FUNCTION_BLOCK Station IMPLEMENTS IStation
VAR_INPUT
END_VAR
VAR_OUTPUT
END_VAR
VAR
	_Clear : BOOL;
	_Complete : BOOL;
	_Operating : BOOL;
	_Ready : BOOL;
	_Positions : ARRAY[1..4] OF MC_LREAL;
	NumberOfPositions : INT;
	AssignedPositions : INT := 1;
	StationMovers : INT;
	_OperationTime : TIME := T#1S;
	Operation : ton;
	_HasMover : BOOL;
END_VAR

IF _HasMover THEN
	_Operating := TRUE;
	_Clear := FALSE;
	_Ready := FALSE;
	Operation.IN := TRUE;
	IF Operation.Q THEN
		_Complete := TRUE;
		IF StationMovers = 0 THEN
			_HasMover := FALSE;
			Operation.IN := FALSE;
		END_IF
	END_IF
ELSE
	_Complete := FALSE;
	_Clear := TRUE;
	_Operating := FALSE;
	_Ready := TRUE;
END_IF

Operation(PT := _OperationTime);

{warning 'add method implementation '}
METHOD HasMover : BOOL
StationMovers := StationMovers + 1;
IF StationMovers = NumberOfPositions THEN
	_HasMover := TRUE;
END_IF
END_METHOD

{warning 'add method implementation '}
METHOD IsClear : BOOL
IsClear := _Clear;
END_METHOD

{warning 'add method implementation '}
METHOD isComplete : BOOL
isComplete := _Complete;
END_METHOD

{warning 'add method implementation '}
METHOD IsOperating : BOOL
IsOperating := _Operating;
END_METHOD

{warning 'add method implementation '}
METHOD IsReady : BOOL
IsReady := _Ready;
END_METHOD

METHOD MoverAway : BOOL
VAR_INPUT
END_VAR
StationMovers := StationMovers - 1;
END_METHOD

{warning 'add property implementation'}
PROPERTY Position : MC_LREAL
GET
Position := _Positions[AssignedPositions];
AssignedPositions := AssignedPositions + 1;
IF AssignedPositions > NumberOfPositions THEN
	AssignedPositions := 1;
END_IF
END_GET
SET
IF NumberOfPositions < 5 THEN
	NumberOfPositions := NumberOfPositions + 1;
	_Positions[NumberOfPositions] := Position;
END_IF
END_SET
END_PROPERTY

PROPERTY TempPropTime : time
GET
TempPropTime := _OperationTime;
END_GET
SET
_OperationTime := TempPropTime;
END_SET
END_PROPERTY

END_FUNCTION_BLOCK

(* stored: Version 1.1.0.1, ProductVersion 3.1.4024.9
   POU Station: Id {c0ea4e62-fbfe-4a62-8def-c1a022a86e9d}, SpecialFunc None
   Method HasMover: Id {5275ace3-94b3-4866-84de-13c179bb6267}
   Method IsClear: Id {8e25d200-227b-4162-a115-dff1d5795336}
   Method isComplete: Id {9f684948-b635-426f-b337-4bc540f41ce6}
   Method IsOperating: Id {e1a11572-f297-45c3-a812-60896aa74d29}
   Method IsReady: Id {c3ad09cd-a86e-4a42-ac30-9f0ab4039334}
   Method MoverAway: Id {4a991ad7-ceff-49bd-89ed-87c906d2b63f}
   Property Position: Id {4add20f7-beba-4a92-8079-611b8f00a59f}
   Get Get: Id {acdae7bd-9c6a-4c62-9baf-3c698e09701d}
   Set Set: Id {c1baf216-d857-42c6-bc5c-effe4378b80c}
   Property TempPropTime: Id {518877d8-6edc-4b69-adf3-92a21d5791e4}
   Get Get: Id {bbcd0dec-698f-451a-acd7-2bf330414c5a}
   Set Set: Id {aec1bbcc-ca82-4261-91fa-a486aafcad09} *)
